(* IEC 61131-3 sources: Caravan/Archiv/12-04-19/Stations/MachineControl/MachineControl/Class/Grid_Class, 1 file *)

(* ---- Grid_Class.st ---- *)
(*!
<Class
	Name               = "Grid_Class"
	Revision           = "0.0"
	RealtimeTask       = "false"
	CyclicTask         = "true"
	DefCyclictime      = "50 ms"
	BackgroundTask     = "false"
	Sigmatek           = "false"
	OSInterface        = "false"
	HighPriority       = "false"
	Automatic          = "false"
	UpdateMode         = "Prescan"
	SharedCommandTable = "true"
	Objectsize         = "(720,480)">
	<Channels>
		<Server Name="ActualAmps_S" Visualized="true" Initialize="false" WriteProtected="false" Retentive="false"/>
		<Server Name="ActualPower_S" Visualized="true" Initialize="false" WriteProtected="false" Retentive="false"/>
		<Server Name="ClassSvr" Visualized="false" Initialize="false" WriteProtected="true" Retentive="false"/>
		<Server Name="MaxSensorAmps_S" Visualized="true" Initialize="false" WriteProtected="false" Retentive="File"/>
		<Server Name="Netzspannung" Visualized="true" Initialize="false" WriteProtected="false" Retentive="File"/>
		<Server Name="ResetKwh_S" Visualized="true" Initialize="false" WriteProtected="false" Retentive="false"/>
		<Server Name="Wattsec_Used_S" Visualized="true" Initialize="false" WriteProtected="false" Retentive="SRam"/>
		<Client Name="ActualAmps_C" Required="true" Internal="false"/>
	</Channels>
</Class>
*)
Grid_Class : CLASS
  //Servers:
	ClassSvr 	: SvrChCmd_DINT;
	ActualAmps_S 	: SvrCh_DINT;
	ActualPower_S 	: SvrCh_DINT;
	MaxSensorAmps_S 	: SvrCh_DINT;
	ResetKwh_S 	: SvrCh_DINT;
	Wattsec_Used_S 	: SvrCh_DINT;
	Netzspannung 	: SvrCh_DINT;
  //Clients:
	ActualAmps_C 	: CltCh_DINT;
  //Variables:
		SectionCounter_VAR 	: DINT;
		SectionPower_VAR 	: DINT;
		OPS_VAR 	: UDINT;
		WattsecAdding_Var 	: DINT;
		PrepValue_VAR 	: DINT;
  //Functions:

	FUNCTION VIRTUAL GLOBAL CyWork
		VAR_INPUT
			EAX 	: UDINT;
		END_VAR
		VAR_OUTPUT
			state (EAX) 	: UDINT;
		END_VAR;
  //Tables:
	FUNCTION @STD
		VAR_OUTPUT
			ret_code	: CONFSTATES;
		END_VAR;
	FUNCTION GLOBAL TAB @CT_;
END_CLASS;

FUNCTION VIRTUAL GLOBAL Grid_Class::CyWork
	VAR_INPUT
		EAX 	: UDINT;
	END_VAR
	VAR_OUTPUT
		state (EAX) 	: UDINT;
	END_VAR

      ActualAmps_C  :=  ActualAmps_C.Read();
      MaxSensorAmps_S :=  MaxSensorAmps_S.Read();
      ResetKwh_S  :=  ResetKwh_S.Read();

       //Keine Division durch 0
       if MaxSensorAmps_S = 0 then

            MaxSensorAmps_S.Write(input:=1);

       end_if;

       //Aktueller Strom errechnen
        ActualAmps_S  :=  ActualAmps_S.Write(input:=(ActualAmps_C*1000) / (10000/MaxSensorAmps_S));

        //Aktuelle Wat berechnen
        ActualPower_S :=  ActualPower_S.Write(input:=(Netzspannung*ActualAmps_S/1000));

        // Stromzähler addieren
        SectionCounter_VAR += 1;
        SectionPower_VAR  +=  ActualPower_S;

        if ops.tAbsolute  >= OPS_VAR + 1000 then

           WattsecAdding_Var  :=  (SectionPower_VAR / SectionCounter_VAR);

           PrepValue_VAR    :=    (WattsecAdding_Var/10) + Wattsec_Used_S;

           Wattsec_Used_S.Write(input:=PrepValue_VAR);

           SectionCounter_VAR :=  0;

           SectionPower_VAR   :=  0;

           OPS_VAR  :=  ops.tAbsolute;

        end_if;

        //Reset KWh
        if ResetKwh_S = 1 then

          Wattsec_Used_S  :=  Wattsec_Used_S.Write(input:=0);

        end_if;

	state := READY;

END_FUNCTION
